INTERFACE ITF_Regelschuif_OutOpen_DG

METHOD set : BOOL
VAR_INPUT
	state : BOOL;
END_VAR
END_METHOD

END_INTERFACE

(* stored: Version 1.1.0.1, ProductVersion 3.1.4026.8
   Itf ITF_Regelschuif_OutOpen_DG: Id {fa9537f2-3d09-42d2-878b-acaf5cfa26c3}
   Method set: Id {9d00375f-c37f-401f-8b1d-5aaac24b2ff6} *)
